FUNCTION_BLOCK DualModuleTmsSwitch EXTENDS MC2_Axis_Base IMPLEMENTS ITF_TmsSwitch
VAR_INPUT
	StateMachine : IPmlStateMachine;
END_VAR
VAR_OUTPUT
END_VAR
VAR
	_exchangeMover : IMover;
	_currentStation : ITF_SwitchStation;
	_demandPosition : MC_LREAL;
	_upPosition : MC_LREAL;
	_middlePosition : MC_LREAL;
	_downPosition : MC_LREAL;
	_SwitchVelocity : MC_LREAL := 100.0;
	arrTrackIds : ARRAY[1..4] OF OTCID;
	stSwitchInfo : TmsSwitchInfo;
END_VAR

{analysis -2}

METHOD Cycle : HRESULT
VAR_INPUT
END_VAR
Cycle := S_OK;
CASE stSwitchInfo.State OF
	TmsSwitchState.Init:
		IF NOT THIS^.hasError() THEN
			stSwitchInfo.State := TmsSwitchState.Ready;
		END_IF
		
	TmsSwitchState.Ready:
		IF StateMachine.GetCurrentState() = E_PMLState.ePMLState_Clearing THEN
			SUPER^.EnableAxis();
			stSwitchInfo.State := TmsSwitchState.Enabling;
		END_IF	
		
	TmsSwitchState.Enabling:
		IF SUPER^.isEnabled() THEN
			stSwitchInfo.State := TmsSwitchState.Enabled;
		END_IF
		
	TmsSwitchState.Enabled:
		IF StateMachine.GetCurrentState() = E_PMLState.ePMLState_Resetting THEN
			IF SUPER^.MoveToPosition(Position := _middlePosition, Velocity := 100.0) OR SUPER^.isAtPosition(position := _middlePosition) THEN
				stSwitchInfo.State := TmsSwitchState.Resetting;
			END_IF
		END_IF
		IF StateMachine.GetCurrentState() = E_PMLState.ePMLState_Aborting
			OR StateMachine.GetCurrentState() = E_PMLState.ePMLState_Stopping THEN
			SUPER^.DisableAxis();
			stSwitchInfo.State := TmsSwitchState.Disabling;
		END_IF
		
	TmsSwitchState.Resetting:
		IF SUPER^.isAtPosition(position := MiddlePosition) THEN
			stSwitchInfo.State := TmsSwitchState.Waiting;
		END_IF	
	
	TmsSwitchState.Waiting:
		IF StateMachine.GetCurrentState() = E_PMLState.ePMLState_Aborting
			OR StateMachine.GetCurrentState() = E_PMLState.ePMLState_Stopping THEN
			SUPER^.DisableAxis();
			stSwitchInfo.State := TmsSwitchState.Disabling;
		END_IF
		
	TmsSwitchState.AssignMover:
		IF HasMover() THEN
			IF FindNewTrack() <> 0 THEN
				stSwitchInfo.State := TmsSwitchState.Moving;
			END_IF
		ELSE
			stSwitchInfo.State := TmsSwitchState.Moving;
		END_IF

	TmsSwitchState.Moving:	
		IF SUPER^.isAtPosition(_demandPosition) THEN
			stSwitchInfo.State := TmsSwitchState.Done;
		END_IF
	
	TmsSwitchState.Done:
		IF _currentStation <> 0 THEN
			IF _currentStation.SwitchMoveComplete() THEN
				_exchangeMover := 0;
				_currentStation := 0;
			END_IF	
		END_IF
		stSwitchInfo.State := TmsSwitchState.Waiting;

	TmsSwitchState.Disabling:
		IF NOT THIS^.isEnabled() THEN
			THIS^.ResetAxis();
			stSwitchInfo.State := TmsSwitchState.Init;
		END_IF
	ELSE
		Cycle := E_FAIL;
END_CASE

//Cyclic get switch info
stSwitchInfo.ActPos := SUPER^._axis.NcToPlc.ActPos;
stSwitchInfo.Position := Switch;

SUPER^.Cycle();
END_METHOD

PROPERTY DownPosition : MC_LREAL
GET
DownPosition := _downPosition;
END_GET
SET
_downPosition := DownPosition;
END_SET
END_PROPERTY

METHOD PUBLIC ExchangeMover : BOOL
VAR_INPUT
	Mover : IMover;
	CurrentStation : ITF_SwitchStation;
END_VAR
IF _exchangeMover = 0 AND stSwitchInfo.State = TmsSwitchState.Waiting AND NOT (stSwitchInfo.Mode = TmsSwitchMode.Manual) THEN
	_exchangeMover := Mover;	
	_currentStation := CurrentStation;
	ExchangeMover := TRUE;
END_IF
END_METHOD

METHOD PUBLIC FindNewTrack : OTCID
VAR_INPUT
END_VAR
VAR
	TmsMoverInterface : ITmsMover;
END_VAR
IF __QUERYINTERFACE(_exchangeMover,TmsMoverInterface) THEN
	IF Switch = TmsSwitchPosition.Up THEN
		IF TmsMoverInterface.ActiveTrack = arrTrackIds[3] THEN
			TmsMoverInterface.ActivateTrack(newTrack := arrTrackIds[1]);
		END_IF
	ELSIF Switch = TmsSwitchPosition.Middle THEN
		IF TmsMoverInterface.ActiveTrack = arrTrackIds[1] THEN
			TmsMoverInterface.ActivateTrack(newTrack := arrTrackIds[3]);
		ELSIF TmsMoverInterface.ActiveTrack = arrTrackIds[2] THEN
			TmsMoverInterface.ActivateTrack(newTrack := arrTrackIds[4]);
		END_IF
	ELSE
		IF TmsMoverInterface.ActiveTrack = arrTrackIds[4] THEN
			TmsMoverInterface.ActivateTrack(newTrack := arrTrackIds[2]);	
		END_IF
	END_IF
END_IF
FindNewTrack := TmsMoverInterface.ActiveTrack;
END_METHOD

METHOD HasMover : BOOL
VAR_INPUT
END_VAR
HasMover := _exchangeMover <> 0;
END_METHOD

PROPERTY PUBLIC MiddlePosition : MC_LREAL
GET
MiddlePosition := _middlePosition;
END_GET
SET
_middlePosition := MiddlePosition;
END_SET
END_PROPERTY

METHOD PUBLIC MoveTo : BOOL
VAR_INPUT
	positionState : TmsSwitchPosition;
END_VAR
CASE positionState OF
	TmsSwitchPosition.Down:
		IF NOT SUPER^.isAtPosition(position := _downPosition) THEN
			IF SUPER^.MoveToPosition(Position := _downPosition, Velocity := _SwitchVelocity) THEN
				MoveTo := TRUE;
				stSwitchInfo.State := TmsSwitchState.AssignMover;
				_demandPosition := _downPosition;
			END_IF
		END_IF	
	TmsSwitchPosition.Middle:
		IF NOT SUPER^.isAtPosition(position := _middlePosition) THEN
			IF SUPER^.MoveToPosition(Position := _middlePosition, Velocity := _SwitchVelocity) THEN
				MoveTo := TRUE;
				stSwitchInfo.State := TmsSwitchState.AssignMover;
				_demandPosition := _middlePosition;
			END_IF
		END_IF	
	TmsSwitchPosition.Up:
		IF NOT SUPER^.isAtPosition(position := _upPosition) THEN
			IF SUPER^.MoveToPosition(Position := _upPosition, Velocity := _SwitchVelocity) THEN
				MoveTo := TRUE;
				stSwitchInfo.State := TmsSwitchState.AssignMover;
				_demandPosition := _upPosition;
			END_IF
		END_IF	
	TmsSwitchPosition.Moving:
		MoveTo := FALSE;
	ELSE
		MoveTo := FALSE;
END_CASE
END_METHOD

METHOD SetAutomaticMode : BOOL
VAR_INPUT
END_VAR
stSwitchInfo.Mode := TmsSwitchMode.Automatic;
END_METHOD

METHOD SetManualMode : BOOL
VAR_INPUT
END_VAR
stSwitchInfo.Mode := TmsSwitchMode.Manual;
END_METHOD

PROPERTY PUBLIC Switch : TmsSwitchPosition
GET
IF SUPER^.isAtPosition(position := _upPosition) THEN
	Switch := TmsSwitchPosition.Up;
ELSIF SUPER^.isAtPosition(position := _middlePosition) THEN
	Switch := TmsSwitchPosition.Middle;
ELSIF SUPER^.isAtPosition(position := _downPosition) THEN
	Switch := TmsSwitchPosition.Down;
ELSE
	Switch := TmsSwitchPosition.Moving;
END_IF
END_GET
END_PROPERTY

PROPERTY SwitchVelocity : MC_LREAL;
GET
SwitchVelocity := _SwitchVelocity;
END_GET
SET
_SwitchVelocity := SwitchVelocity;
END_SET
END_PROPERTY

PROPERTY TrackIds : array[1..4] of otcid
GET
TrackIds := arrTrackIds;
END_GET
SET
arrTrackIds := TrackIds;
END_SET
END_PROPERTY

PROPERTY PUBLIC UpperPosition : MC_LREAL
GET
UpperPosition := _upPosition;
END_GET
SET
_upPosition := UpperPosition;
END_SET
END_PROPERTY

END_FUNCTION_BLOCK

(* stored: Version 1.1.0.1, ProductVersion 3.1.4024.12
   POU DualModuleTmsSwitch: Id {b99b16cd-cff3-4deb-90c3-1a32a82a4df9}, SpecialFunc None
   Method Cycle: Id {87873dec-7b42-4805-90b6-759ce824ebea}
   Property DownPosition: Id {599e43c8-9e54-4127-98c0-830d987c6670}
   Get Get: Id {d576d882-31e3-4df4-8d25-fb96bcb31534}
   Set Set: Id {52d02993-45ed-4cc1-b7c9-7e50079230a8}
   Method ExchangeMover: Id {55ccaa02-7858-4213-8d05-433f72c712e6}
   Method FindNewTrack: Id {f8facd12-02a9-4323-9c07-28752afef02e}
   Method HasMover: Id {0c44fa73-b6c5-42b1-9f3a-b9c3b353571a}
   Property MiddlePosition: Id {a5913fe6-4718-4392-9be8-d67930c5a069}
   Get Get: Id {4ade54e3-8b33-4ead-b3b1-391afaf4c4b3}
   Set Set: Id {6ffe5ecb-8591-417d-81eb-1b6851de2312}
   Method MoveTo: Id {1257cc6d-b02a-46ca-8efb-e12582dbd46c}
   Method SetAutomaticMode: Id {5d2127ff-7894-4041-9880-78681ac45ab3}
   Method SetManualMode: Id {b1c41df0-1df7-4794-ab5d-918311a70b04}
   Property Switch: Id {0b7e1326-662c-4bc8-a99b-c301c7bc3754}
   Get Get: Id {6caed8c1-8918-4b95-8833-b1d3db921a19}
   Property SwitchVelocity: Id {23d2c69c-54c3-4033-bf24-addeee1198d3}
   Get Get: Id {63c4a6c5-28c8-403b-828f-bffb40704c3b}
   Set Set: Id {a0f07dce-a6c5-4f13-a413-55d73aacfb92}
   Property TrackIds: Id {297989bc-9ff5-412a-89d0-1e0ef6098068}
   Get Get: Id {721632d5-47ed-4060-a975-8bc16c5085ad}
   Set Set: Id {cc05dbf6-96b3-41b2-9fa2-61c5be84c081}
   Property UpperPosition: Id {d1dd9c15-1bcf-4557-9ed1-65e173a50daa}
   Get Get: Id {b1aa855a-5521-476e-a12b-14a1c1a88b2a}
   Set Set: Id {f811094b-d3fc-4924-bea3-35ccbae64bb4} *)
